// TIA Portal V18 export
FUNCTION_BLOCK "HMI_In_selection_handling"   // FB4, SCL
{ S7_Optimized_Access := 'FALSE' }
VERSION : 0.1
// stored: AutoNumber true, IsIECCheckEnabled false, SetENOAutomatically false, UDAEnableTagReadback false
   VAR_INPUT
      step_size : Int := 50;
      Timer_duration : Time := T#1s;
      Time_pulse_speed : Time := T#1ms;
   END_VAR
   VAR_IN_OUT
      variable : Int;
   END_VAR
BEGIN


   IF "Rising_edge_next".Q THEN
       "Rising_edge_next".Q := 0;
       #variable := #variable + #step_size;
   END_IF;

   IF "Rising_edge_prev".Q THEN
       "Rising_edge_prev".Q := 0;
       #variable := #variable - #step_size;
       #variable := MAX(IN1 := #variable, IN2 := 0);
   END_IF;

   IF "Rising_edge_enter".Q THEN
       "Rising_edge_enter".Q := 0;
       "Var_HMI".in_selection := 0;
       "Var_HMI".selection_no := 0;

   END_IF;

   "IEC_Timer_0_DB_22".TON(IN:="NEXT_Button" OR "PREV_Button",
                           PT:=#Timer_duration);


   IF "IEC_Timer_0_DB_22".Q THEN


       "IEC_Timer_0_DB_16".TP(IN := "Clock_10Hz",
                              PT := #Time_pulse_speed);

       IF "IEC_Timer_0_DB_16".Q THEN

           IF "NEXT_Button" THEN
               #variable := #variable + 100;
           END_IF;

           IF "PREV_Button" THEN
               #variable := #variable - 100;
               #variable := MAX(IN1 := #variable, IN2 := 0);
           END_IF;

       END_IF;

       END_IF;


       IF NOT "NEXT_Button" AND NOT "PREV_Button" THEN
           RESET_TIMER("IEC_Timer_0_DB_22");
       END_IF;
END_FUNCTION_BLOCK
